// SIMATIC S7-200 project (STEP 7-Micro/WIN), CPU 221 REL 01.10

SYMBOL_TABLE USER1
START            I0.0
STOPP            I0.1
D1               Q0.0
D2               Q0.1
D3               Q0.2
D4               Q0.3
D5               Q0.4
D6               Q0.5
D7               Q0.6
D8               Q0.7
END_SYMBOL_TABLE

ORGANIZATION_BLOCK MAIN:OB1
TITLE=PROGRAM COMMENTS
BEGIN
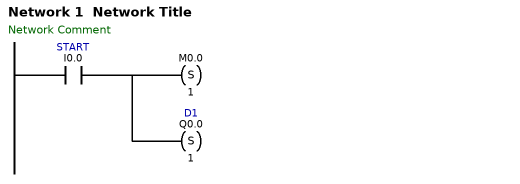
Network 1 // Network Title
// Network Comment
LD     START:I0.0
S      M0.0, 1
S      D1:Q0.0, 1
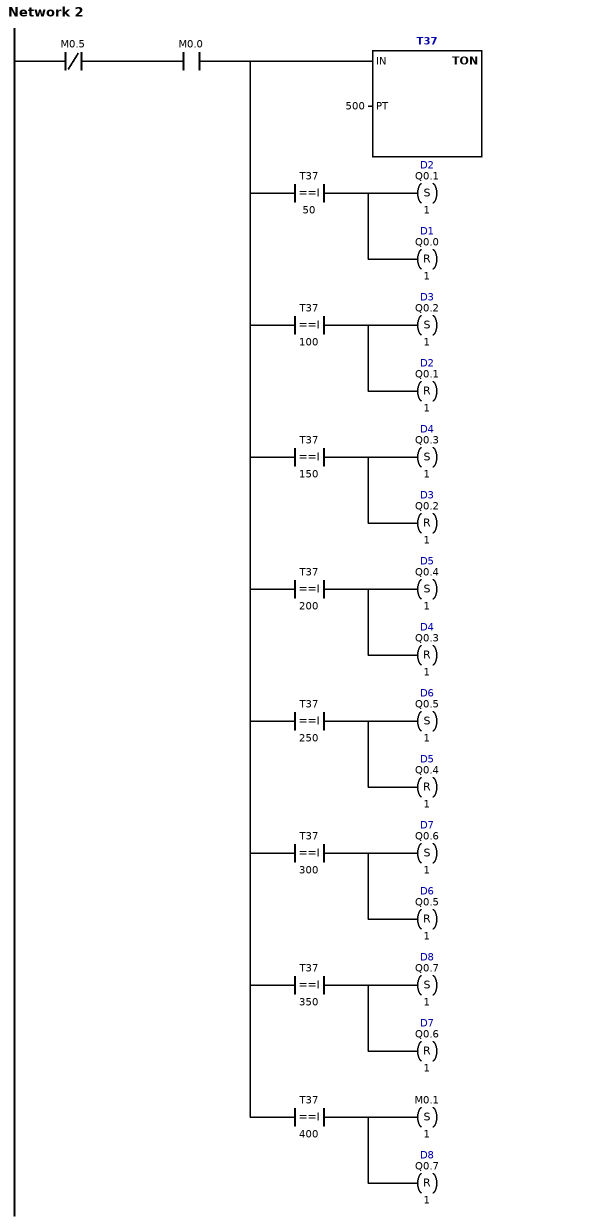
Network 2
LDN    M0.5
A      M0.0
LPS
TON    T37, 500
AW=    T37, 50
S      D2:Q0.1, 1
R      D1:Q0.0, 1
LRD
AW=    T37, 100
S      D3:Q0.2, 1
R      D2:Q0.1, 1
LRD
AW=    T37, 150
S      D4:Q0.3, 1
R      D3:Q0.2, 1
LRD
AW=    T37, 200
S      D5:Q0.4, 1
R      D4:Q0.3, 1
LRD
AW=    T37, 250
S      D6:Q0.5, 1
R      D5:Q0.4, 1
LRD
AW=    T37, 300
S      D7:Q0.6, 1
R      D6:Q0.5, 1
LRD
AW=    T37, 350
S      D8:Q0.7, 1
R      D7:Q0.6, 1
LPP
AW=    T37, 400
S      M0.1, 1
R      D8:Q0.7, 1
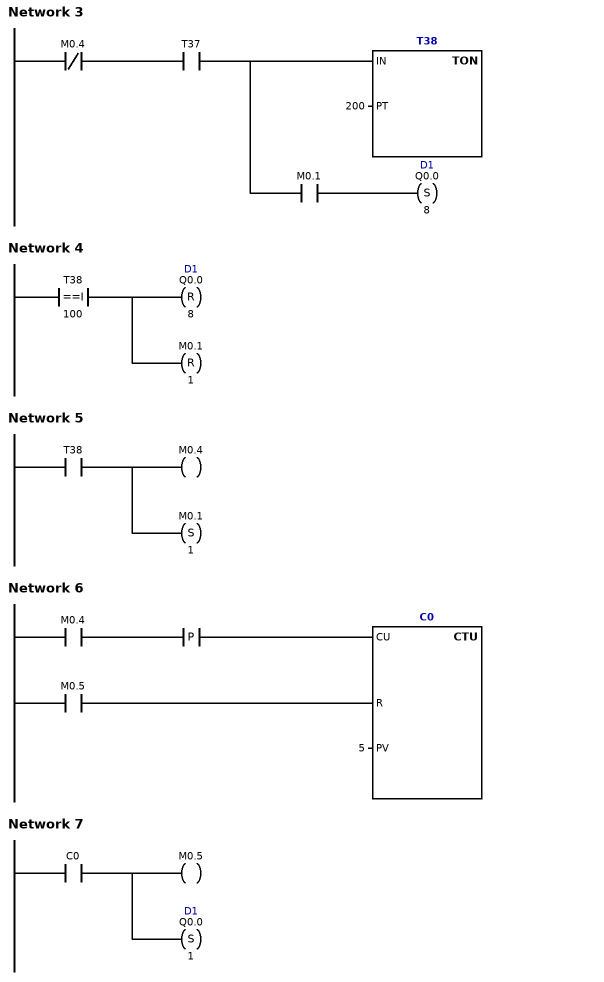
Network 3
LDN    M0.4
A      T37
TON    T38, 200
A      M0.1
S      D1:Q0.0, 8
Network 4
LDW=   T38, 100
R      D1:Q0.0, 8
R      M0.1, 1
Network 5
LD     T38
=      M0.4
S      M0.1, 1
Network 6
LD     M0.4
EU
LD     M0.5
CTU    C0, 5
Network 7
LD     C0
=      M0.5
S      D1:Q0.0, 1
END_ORGANIZATION_BLOCK
